/// <summary>
    /// 
    /// Die PAProcessFunction wickelt einen ACMethod-Aufruf asynchron ab. 
    /// Instanzen von PAProcessFunction werden immer unterhalb von ACComponent der Model- oder VarioBatch-Welt erzeugt.
    /// 
    /// Es gibt drei Varianten der Implementierung
    /// 1. Direkte Ableitung in Form einer asynchronen Prozessfunktion (z.B. PAFDosing, PAFMixing) 
    ///    Nur einmal Instanziierbar (Meist mit Kopplung an Hardware/SPS)
    /// 2. Verwendung der Ableitung PWProcessFunction als Workflow (weitere Info siehe in PWProcessFunction.cs)
    /// 3. Direkte Ableitung als mehrfach Instanziierbar. Beispiel (abstract):
    /// SAPSchnittstelle : ACComponent (Modeltree)
    ///     SAPExport : PAProcessFunction   (Dynamische Instanzen beim SAPSchnittstelle.Exportstart)
    ///     SAPImport : PAProcessFunction   (Dynamische Instanzen beim SAPSchnittstelle.Importstart)
    /// 
    /// Die Statusfolge und die Steuerung von außen ist an die S88 angelehnt
    /// https://www.isa.org/pdfs/microsites121/s-880001/
    /// Methoden zur Steuerung von außen: 
    /// -Start(acMethod)    Starten/Initialisieren des Prozesses
    /// -Run()              Aktivieren des Prozesses
    /// -Pause()            Pausieren des Prozesses
    /// -Resume()           Fortsetzen nach dem Pausieren
    /// -Hold()             Anhalten des Prozesses (längere Pause)
    /// -Restart()          Anfahren nach längerer Pause
    /// -Abort()            Abbrechen des Prozesses
    /// -Stop()             Stoppen des Prozesses
    /// -Reset()            Wechsel in den Grundzustand SMIdle
    /// 
    ///     ACState     | Auto-Next-State  |                |                                               TRANSITION-METHODS
    ///               	|   (No Method)    |   Start()	    |   Run()	    |   Pause()	    |   Resume()	|   Hold()	    |   Restart()	|   Abort()	    |   Stopp()	    |   Reset()
    /// ___________________________________________________________________________________________________________________________________________________________________________________
    /// 
    /// SMIdle		    |           		|  SMStarting   |				|               |               |               |               |               |               |         
    /// -----------------------------------------------------------------------------------------------------------------------------------------------------------------------------------
    /// SMStarting	    |       			|	    		|	SMRunning	|	            |               |               |               |               |               |   SMResetting
    /// -----------------------------------------------------------------------------------------------------------------------------------------------------------------------------------
    /// SMRunning	    | SMCompleted		|               |               | SMPausing		|               | SMHolding	    |	            |  SMAborting   |	SMStopping	|
    /// -----------------------------------------------------------------------------------------------------------------------------------------------------------------------------------
    /// SMCompleted	    |					|               |               |               |               |               |               |               |               |	SMResetting
    /// -----------------------------------------------------------------------------------------------------------------------------------------------------------------------------------
    /// SMResetting	    | SMIdle			|               |               |               |               |               |               |               |               |					
    /// ___________________________________________________________________________________________________________________________________________________________________________________
    /// SMPausing	    | SMPaused			|               |               |               |               |               |               |               |               |					
    /// -----------------------------------------------------------------------------------------------------------------------------------------------------------------------------------
    /// SMPaused		|                   |               |               |               |  SMResuming	|               |               |  SMAborting	|   SMStopping  |	
    /// -----------------------------------------------------------------------------------------------------------------------------------------------------------------------------------
    /// SMResuming	    | SMRunning			|               |               |               |               |               |               |               |               |					
    /// ___________________________________________________________________________________________________________________________________________________________________________________
    /// SMHolding	    | SMHeld			|               |               |               |               |               |               |               |               |					
    /// -----------------------------------------------------------------------------------------------------------------------------------------------------------------------------------
    /// SMHeld			|			        |               |               |               |               |               |SMRestarting	|   SMAborting	|   SMStopping	|
    /// -----------------------------------------------------------------------------------------------------------------------------------------------------------------------------------
    /// SMRestarting	| SMRunning			|               |               |               |               |               |               |               |               |				
    /// ___________________________________________________________________________________________________________________________________________________________________________________
    /// SMAborting	    | SMAborted			|               |               |               |               |               |               |               |               |										
    /// -----------------------------------------------------------------------------------------------------------------------------------------------------------------------------------
    /// SMAborted		|					|               |               |               |               |               |               |               |               |	SMResetting
    /// ___________________________________________________________________________________________________________________________________________________________________________________
    /// SMStopping	    | SMStopped			|               |               |               |               |               |               |               |               |				
    /// -----------------------------------------------------------------------------------------------------------------------------------------------------------------------------------
    /// SMStopped		|					|               |               |               |               |               |               |               |               |	SMResetting
    /// -----------------------------------------------------------------------------------------------------------------------------------------------------------------------------------
    /// </summary>
FUNCTION_BLOCK PAProcessFunction EXTENDS PAClassAlarmingBase IMPLEMENTS IPAProcessFunction
VAR_INPUT
END_VAR
VAR_OUTPUT
END_VAR
VAR
	_Malfunction : PANotifyState;
	_AckMalfunction : BOOL;
END_VAR
VAR PERSISTENT
	_ACState : ACStateEnum;
	_TMMethod : TMMethod;
END_VAR

METHOD PUBLIC Abort : BOOL
VAR_INPUT
END_VAR
IF NOT IsEnabledAbort THEN
	Abort := FALSE;
	RETURN;
END_IF
ACState := ACStateEnum.SMAborting;
Abort := TRUE;
END_METHOD

{attribute 'monitoring' := 'call'}
//{attribute 'TcRpcEnable'}
PROPERTY PUBLIC AckMalfunction : BOOL
GET
AckMalfunction := _AckMalfunction;
END_GET
SET
_AckMalfunction := AckMalfunction;
Root.OnPropertyChangedBool(THIS^, 15, _AckMalfunction);
END_SET
END_PROPERTY

PROPERTY PUBLIC ACMethod : IACMethod
GET
END_GET
END_PROPERTY

{attribute 'monitoring' := 'call'}
//{attribute 'TcRpcEnable'}
PROPERTY PUBLIC ACState : ACStateEnum
GET
ACState := _ACState;
END_GET
SET
_ACState := ACState;
Root.OnPropertyChangedInt(THIS^, 13, _ACState);
END_SET
END_PROPERTY

METHOD PUBLIC FB_postinit
VAR_INPUT
		root : IACVariobatch;
END_VAR
SUPER^.FB_postinit(root);
root.OnPropertyChangedInt(THIS^, 13, _ACState);
root.OnPropertyChangedInt(THIS^, 14, _Malfunction);
root.OnPropertyChangedBool(THIS^, 15, _AckMalfunction);
END_METHOD

METHOD PROTECTED HandleACState
VAR_INPUT
END_VAR
CASE _ACState OF
	ACStateEnum.SMIdle:
		SMIdle();
	ACStateEnum.SMStarting:
		SMStarting();
	ACStateEnum.SMRunning:
		SMRunning();
	ACStateEnum.SMCompleted:
		SMCompleted();
	ACStateEnum.SMResetting:
		SMResetting();
	ACStateEnum.SMPausing:
		SMPausing();
	ACStateEnum.SMPaused:
		SMPaused();
	ACStateEnum.SMResuming:
		SMResuming();
	ACStateEnum.SMHolding:
		SMHolding();
	ACStateEnum.SMHeld:
		SMHeld();
	ACStateEnum.SMRestarting:
		SMRestarting();
	ACStateEnum.SMAborting:
		SMAborting();
	ACStateEnum.SMAborted:
		SMAborted();
	ACStateEnum.SMStopping:
		SMStopping();
	ACStateEnum.SMStopped:
		SMStopped();
END_CASE
END_METHOD

METHOD PROTECTED HandleTMMethod
VAR_INPUT
END_VAR
CASE _TMMethod OF
	TMMethod.TMNone:
		RETURN;
	TMMethod.TMStart :
		Start();
	TMMethod.TMRun:
		Run();
	TMMethod.TMPause:
		Pause();
	TMMethod.TMResume:
		Resume();
	TMMethod.TMHold:
		Hold();
	TMMethod.TMRestart:
		Restart();
	TMMethod.TMAbort:
		Abort();
	TMMethod.TMStopp:
		Stopp();
	TMMethod.TMReset:
		Reset();
END_CASE
_TMMethod := TMMethod.TMNone;
END_METHOD

METHOD PUBLIC Hold : BOOL
VAR_INPUT
END_VAR
IF NOT IsEnabledHold THEN
	Hold := FALSE;
	RETURN;
END_IF
ACState := ACStateEnum.SMHolding;
Hold := TRUE;
END_METHOD

METHOD PUBLIC InvokeSetterBool
VAR_INPUT
	PropertyID : INT;
	PropertyValue : BOOL;
END_VAR
SUPER^.InvokeSetterBool(PropertyID, PropertyValue);
IF PropertyID = 15 THEN
	THIS^.AckMalfunction := PropertyValue;
END_IF
END_METHOD

METHOD PUBLIC InvokeSetterEnum
VAR_INPUT
	PropertyID : INT;
	PropertyValue : INT;
END_VAR
SUPER^.InvokeSetterEnum(PropertyID, PropertyValue);
IF PropertyID = 13 THEN
	THIS^.ACState := PropertyValue;
ELSIF PropertyID = 14 THEN	
	THIS^.Malfunction := PropertyValue;
END_IF
END_METHOD

PROPERTY PUBLIC IsEnabledAbort : BOOL
GET
IsEnabledAbort := _ACState = ACStateEnum.SMRunning OR _ACState = ACStateEnum.SMHeld OR _ACState = ACStateEnum.SMPaused;
END_GET
END_PROPERTY

PROPERTY PUBLIC IsEnabledHold : BOOL
GET
IsEnabledHold := _ACState = ACStateEnum.SMRunning;
END_GET
END_PROPERTY

PROPERTY PUBLIC IsEnabledPause : BOOL
GET
IsEnabledPause := _ACState = ACStateEnum.SMRunning;
END_GET
END_PROPERTY

PROPERTY PUBLIC IsEnabledReset : BOOL
GET
IsEnabledReset := _ACState = ACStateEnum.SMStarting OR _ACState = ACStateEnum.SMCompleted OR _ACState = ACStateEnum.SMAborted OR _ACState = ACStateEnum.SMStopped OR _ACState = ACStateEnum.SMIdle;
END_GET
END_PROPERTY

PROPERTY PUBLIC IsEnabledRestart : BOOL
GET
IsEnabledRestart := _ACState = ACStateEnum.SMHeld;
END_GET
END_PROPERTY

PROPERTY PUBLIC IsEnabledResume : BOOL
GET
IsEnabledResume := _ACState = ACStateEnum.SMPaused;
END_GET
END_PROPERTY

PROPERTY PUBLIC IsEnabledRun : BOOL
GET
IsEnabledRun := _ACState = ACStateEnum.SMStarting;
END_GET
END_PROPERTY

PROPERTY PUBLIC IsEnabledStart : BOOL
GET
IF _ACState = ACStateEnum.SMIdle THEN
		IsEnabledStart := TRUE;
	RETURN;
END_IF
IsEnabledStart := ACMethod.IsValid;
END_GET
END_PROPERTY

PROPERTY PUBLIC IsEnabledStopp : BOOL
GET
IsEnabledStopp := _ACState = ACStateEnum.SMRunning OR _ACState = ACStateEnum.SMHeld OR _ACState = ACStateEnum.SMPaused;
END_GET
END_PROPERTY

{attribute 'monitoring' := 'call'}
//{attribute 'TcRpcEnable'}
PROPERTY PUBLIC Malfunction : PANotifyState
GET
Malfunction := _Malfunction;
END_GET
SET
_Malfunction := Malfunction;
Root.OnPropertyChangedInt(THIS^, 14, _Malfunction);
END_SET
END_PROPERTY

METHOD OnInitMemory
VAR_INPUT
		root : IACVariobatch;
END_VAR
RegisterProperty(root, 13, GCL.cSizeINT); // _ACState
RegisterProperty(root, 14, GCL.cSizeINT); // _Malfunction
RegisterProperty(root, 15, GCL.cSizeBYTE); // _AckMalfunction
SUPER^.OnInitMemory(root);
END_METHOD

METHOD PROTECTED OnMainEnter
VAR_INPUT
END_VAR

VAR
	TMNone: INT;
END_VAR
HandleTMMethod();
HandleACState();
END_METHOD

METHOD PUBLIC Pause : BOOL
VAR_INPUT
END_VAR
IF NOT IsEnabledPause THEN
	Pause := FALSE;
	RETURN;
END_IF
ACState := ACStateEnum.SMPausing;
Pause := TRUE;
END_METHOD

METHOD PUBLIC Reset : BOOL
VAR_INPUT
END_VAR
IF NOT IsEnabledReset THEN
	Reset := FALSE;
	RETURN;
END_IF
ACState := ACStateEnum.SMResetting;
Reset := TRUE;
END_METHOD

METHOD PUBLIC Restart : BOOL
VAR_INPUT
END_VAR
IF NOT IsEnabledRestart THEN
	Restart := FALSE;
	RETURN;
END_IF
ACState := ACStateEnum.SMRestarting;
Restart := TRUE;
END_METHOD

METHOD PUBLIC Resume : BOOL
VAR_INPUT
END_VAR
IF NOT IsEnabledResume THEN
	Resume := FALSE;
	RETURN;
END_IF
ACState := ACStateEnum.SMResuming;
Resume := TRUE;
END_METHOD

METHOD PUBLIC Run : BOOL
VAR_INPUT
END_VAR
IF NOT IsEnabledRun THEN
	Run := FALSE;
	RETURN;
END_IF
ACState := ACStateEnum.SMRunning;
Run := TRUE;
END_METHOD

METHOD PROTECTED SMAborted
VAR_INPUT
END_VAR
END_METHOD

METHOD PROTECTED SMAborting
VAR_INPUT
END_VAR
END_METHOD

METHOD PROTECTED SMCompleted
VAR_INPUT
END_VAR
END_METHOD

METHOD PROTECTED SMHeld
VAR_INPUT
END_VAR
END_METHOD

METHOD PROTECTED SMHolding
VAR_INPUT
END_VAR
END_METHOD

METHOD PROTECTED SMIdle
VAR_INPUT
END_VAR
END_METHOD

METHOD PROTECTED SMPaused
VAR_INPUT
END_VAR
END_METHOD

METHOD PROTECTED SMPausing
VAR_INPUT
END_VAR
END_METHOD

METHOD PROTECTED SMResetting
VAR_INPUT
END_VAR
END_METHOD

METHOD PROTECTED SMRestarting
VAR_INPUT
END_VAR
END_METHOD

METHOD PROTECTED SMResuming
VAR_INPUT
END_VAR
END_METHOD

METHOD PROTECTED SMRunning
VAR_INPUT
END_VAR
END_METHOD

METHOD PROTECTED SMStarting
VAR_INPUT
END_VAR
END_METHOD

METHOD PROTECTED SMStopped
VAR_INPUT
END_VAR
END_METHOD

METHOD PROTECTED SMStopping
VAR_INPUT
END_VAR
END_METHOD

METHOD PUBLIC Start : BOOL
VAR_INPUT
END_VAR
IF NOT IsEnabledStart THEN
		Start := FALSE;
	RETURN;
END_IF
ACState := ACStateEnum.SMRunning;
Start := TRUE;
END_METHOD

METHOD PUBLIC Stopp : BOOL
VAR_INPUT
END_VAR
IF NOT IsEnabledStopp THEN
	Stopp := FALSE;
	RETURN;
END_IF
ACState := ACStateEnum.SMStopping;
Stopp := TRUE;
END_METHOD

END_FUNCTION_BLOCK

(* stored: Version 1.1.0.1, ProductVersion 3.1.4024.6
   POU PAProcessFunction: Id {79b850f6-1962-463e-9639-bcb04767e56d}, SpecialFunc None
   Folder IsEnabledMethods: Id {ab4fa63a-cfbc-4409-bb53-e54781e40a0d}
   Folder Properties: Id {981846ba-357f-4ae5-860a-f032b7423ae9}
   Folder StateMethods: Id {39513048-fbf1-4443-81c5-9efb2ab082af}
   Folder TransitionMethods: Id {dd848e1b-49b8-4b6b-94dc-3a8403668558}
   Method Abort: Id {c9d3ea8d-1551-48d6-9adc-177f5e196019}
   Property AckMalfunction: Id {541a44e3-be9c-41ed-b44d-06cce1c76469}
   Get Get: Id {987b8645-86d8-4d2e-9c74-2f211f3fc0df}
   Set Set: Id {683ffd67-0007-4b68-ae6f-9b0d9eafb8eb}
   Property ACMethod: Id {03d6abe1-7d4c-40d0-acae-55c66cd24e22}
   Get Get: Id {5573962a-f6f7-42f4-bdc2-d4c3e6f57f25}
   Property ACState: Id {2bfb6a4f-c65f-464b-a0a9-6a2a61d70739}
   Get Get: Id {48811ade-1d01-4881-a302-7d66db477b79}
   Set Set: Id {4a09b30d-1c54-4c7a-8f6a-b88792a318c6}
   Method FB_postinit: Id {0dd89ec2-265b-4a09-90ed-a83b2f79da3c}
   Method HandleACState: Id {b88d4a9d-bbae-4757-bd10-06754fb1d11a}
   Method HandleTMMethod: Id {853bc94c-8941-4e51-a75b-bb32a89a55da}
   Method Hold: Id {d06ffbbb-aed6-47cf-8854-4c72fb7f13a7}
   Method InvokeSetterBool: Id {928e2a59-abc6-4878-8149-162c5c587f62}
   Method InvokeSetterEnum: Id {ebe13666-0bec-4a12-b3f6-b455fb3fa089}
   Property IsEnabledAbort: Id {809f95e9-ef40-4837-b3ab-319b6e4d2710}
   Get Get: Id {821b2a7d-3dfc-407c-ba97-8b53abeb18b5}
   Property IsEnabledHold: Id {1aa723e4-4ed9-4039-959d-ac484328df09}
   Get Get: Id {80eac49d-e380-49f9-baf8-86297410ecbe}
   Property IsEnabledPause: Id {64f0fee1-afd3-4727-9247-2be165d423a2}
   Get Get: Id {628b572a-4b4a-45b6-9d4d-3f9e72a721a5}
   Property IsEnabledReset: Id {2adcf514-1621-4801-b3e1-7d337c81f8bf}
   Get Get: Id {723366dc-c509-4dbc-9827-de2e90b0fbe6}
   Property IsEnabledRestart: Id {76f78737-2cd6-4463-b1fd-070d9f04c98b}
   Get Get: Id {b564b76a-5521-493f-a77f-5da63164d795}
   Property IsEnabledResume: Id {d0b55608-2a49-4284-b7d2-02796330be3f}
   Get Get: Id {c4abcf28-688c-4e42-b855-9f905f6e699a}
   Property IsEnabledRun: Id {ea60c16f-f0f6-4148-9902-b84c357ea5f1}
   Get Get: Id {e7441336-7751-44cd-8445-87605087d421}
   Property IsEnabledStart: Id {7fbc58a0-0333-4f8a-ad36-8dc5b9cf6667}
   Get Get: Id {c3715939-474e-4b23-b373-2bfb98a2c585}
   Property IsEnabledStopp: Id {d68ba562-f1f2-48de-b8c2-92f232e7f4a7}
   Get Get: Id {1043286c-0718-40ba-87fd-90b323b177c6}
   Property Malfunction: Id {902523fc-57ed-4777-823a-f58e643c1c2d}
   Get Get: Id {abb53ce4-c1c4-4a6d-aab5-909f2ed3922d}
   Set Set: Id {60b074b9-dd02-4fd8-8ee9-e4041f301c72}
   Method OnInitMemory: Id {5ba8255f-96c2-4bfa-a9e4-eed2a16005cf}
   Method OnMainEnter: Id {133bba2a-5ec4-42cf-99b8-5a804abd5fa6}
   Method Pause: Id {b4bfe6a4-0adc-4b89-aecd-c90778d5a8af}
   Method Reset: Id {ad9e6810-26b8-4a7b-b6dd-fc3819d565de}
   Method Restart: Id {2d9d79d6-4691-4a1b-b2a0-e74fdbdc5a75}
   Method Resume: Id {58a328c9-cfef-4ef2-b8b3-28de79d296bb}
   Method Run: Id {d030c7db-8a24-4166-89cc-95cfcddda6e8}
   Method SMAborted: Id {206a6db6-6022-4454-889c-0fc156ec2929}
   Method SMAborting: Id {fcc3d314-b6fe-4082-8539-c0fd8c65df3c}
   Method SMCompleted: Id {bc125f72-fa83-490c-9187-1c0ecd739724}
   Method SMHeld: Id {6c78f470-57ab-4fa7-9361-76d84bdcd577}
   Method SMHolding: Id {fa8573d4-a549-4bc4-9d7e-c2af3ed33271}
   Method SMIdle: Id {7065863c-db7c-46bc-84d4-71be823c84c8}
   Method SMPaused: Id {06ec23ff-9bb0-4472-b19b-be5240dec765}
   Method SMPausing: Id {85caec46-008a-410e-9137-60d12f575c1c}
   Method SMResetting: Id {2bd66971-b68e-4df2-abb5-3be18009cf3a}
   Method SMRestarting: Id {64e4fe97-2495-4ad1-9e58-6ae21d343cf7}
   Method SMResuming: Id {d65c255f-866b-48ea-8598-1470e12d5d07}
   Method SMRunning: Id {feeb4b25-34c8-4a76-ac47-2878d29d7c52}
   Method SMStarting: Id {6e11f845-1709-4c24-8591-6696212a45b8}
   Method SMStopped: Id {fb806c1a-a32e-40ca-b70c-ff2b8b5a4e17}
   Method SMStopping: Id {a4bfcb26-d76e-4f0f-b940-e96e92ba6a4b}
   Method Start: Id {0f87f056-075c-4224-8528-1c9a24f52cf5}
   Method Stopp: Id {7f82a9aa-c4ef-44ff-ae83-d23bf796f23b} *)
